(* IEC 61131-3 sources: RAG_PLC/data/result/test/003, 2 files *)

(* ---- wrapped.st ---- *)
(* =========================================================
   Generated by PLC-Eval Benchmark Wrapper
   ========================================================= *)

FUNCTION_BLOCK LLM_Wrapper_FB
VAR_INPUT
	T : REAL;  // 温度 (°C)
	RN : REAL; // 参考电阻值 (Ω)
	B : REAL;  // 负温度系数 (1/°C)
END_VAR

VAR_OUTPUT
	RES_NTC : REAL;  // 计算得到的电阻值 (Ω)
END_VAR

RES_NTC := RN * EXP(B * (1.0 / (T + 273.15) - 1.0 / (25.0 + 273.15)));
END_FUNCTION_BLOCK

PROGRAM Auto_Proxy_Prg
  VAR
    instance : LLM_Wrapper_FB;
  END_VAR

  instance();
END_PROGRAM

CONFIGURATION Config0
  RESOURCE Res0 ON PLC
    TASK TaskMain(INTERVAL := T#20ms, PRIORITY := 0);
    PROGRAM Inst0 WITH TaskMain : Auto_Proxy_Prg;
  END_RESOURCE
END_CONFIGURATION

(* ---- raw_code.st ---- *)
VAR_INPUT
	T : REAL;  // 温度 (°C)
	RN : REAL; // 参考电阻值 (Ω)
	B : REAL;  // 负温度系数 (1/°C)
END_VAR

VAR_OUTPUT
	RES_NTC : REAL;  // 计算得到的电阻值 (Ω)
END_VAR

RES_NTC := RN * EXP(B * (1.0 / (T + 273.15) - 1.0 / (25.0 + 273.15)));
